{attribute 'pack_mode' := '2'}
TYPE ST_STATION_STATE :
STRUCT
  State           : E_STATION_STATE;
  {attribute 'displaymode':='bin'}
  nMask           : BYTE;
  nMoverId        : USINT;
  rMoverModPos    : LREAL;            // modulo position of detected mover
  nQueue          : USINT;            // queue count for station
END_STRUCT
END_TYPE

(* stored: Version 1.1.0.1, ProductVersion 3.1.4026.18
   DUT ST_STATION_STATE: Id {87b7b128-9986-420c-b5d3-f350cbe78799} *)
